Staubli VAL3: primeMotStack.pgx

program primeMotStack()
begin
  //!brief
  //Prime the motion stack monitor
  bDisplayed=false
  // set timer for motion stack monitoring
  tmMotionStack=clock()
end
